// Mitsubishi GX Works2 project: plc_program   PLC: FX1N/FX1NC

PROGRAM MAIN
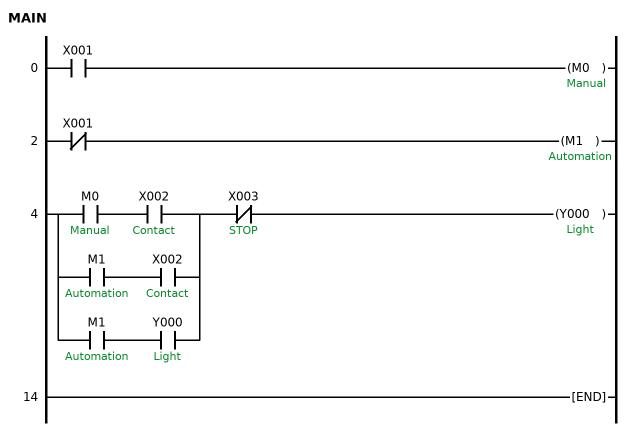
0     LD      X001
      OUT     M0  ; Manual
2     LDI     X001
      OUT     M1  ; Automation
4     LD      M0  ; Manual
      AND     X002  ; Contact
      LD      M1  ; Automation
      AND     X002  ; Contact
      ORB
      LD      M1  ; Automation
      AND     Y000  ; Light
      ORB
      ANI     X003  ; STOP
      OUT     Y000  ; Light
14    END
END_PROGRAM
